(* IEC 61131-3 sources: Std_PalletMover/Class/EncoderpulsesToDegrees, 1 file *)

(* ---- EncoderpulsesToDegrees.st ---- *)
(*!
<Class
	Name               = "EncoderpulsesToDegrees"
	Revision           = "0.0"
	RealtimeTask       = "false"
	CyclicTask         = "true"
	BackgroundTask     = "false"
	Sigmatek           = "false"
	OSInterface        = "false"
	HighPriority       = "false"
	Automatic          = "false"
	UpdateMode         = "Prescan"
	SharedCommandTable = "true"
	Objectsize         = "(512,120)">
	<Channels>
		<Server Name="ClassSvr" Visualized="false" Initialize="false" WriteProtected="true" Retentive="false"/>
		<Server Name="Degrees" Visualized="false" Initialize="false" WriteProtected="true" Retentive="false"/>
		<Server Name="GearRatio" Visualized="false" Initialize="true" WriteProtected="false" Retentive="false"/>
		<Server Name="PulsesPerRound" Visualized="false" Initialize="true" WriteProtected="false" Retentive="false"/>
		<Client Name="EncoderPulses" Required="false" Internal="false"/>
	</Channels>
</Class>
*)
EncoderpulsesToDegrees : CLASS
  //Servers:
	ClassSvr 	: SvrChCmd_DINT;
	PulsesPerRound 	: SvrCh_REAL;
	GearRatio 	: SvrCh_REAL;
	Degrees 	: SvrCh_REAL;
  //Clients:
	EncoderPulses 	: CltCh_DINT;
  //Variables:
  //Functions:

	FUNCTION VIRTUAL GLOBAL CyWork
		VAR_INPUT
			EAX 	: UDINT;
		END_VAR
		VAR_OUTPUT
			state (EAX) 	: UDINT := READY;
		END_VAR;

	FUNCTION VIRTUAL GLOBAL Degrees::Read
		VAR_OUTPUT
			output (EAX) 	: REAL;
		END_VAR;
  //Tables:
	FUNCTION @STD
		VAR_OUTPUT
			ret_code	: CONFSTATES;
		END_VAR;
	FUNCTION GLOBAL TAB @CT_;
END_CLASS;

FUNCTION VIRTUAL GLOBAL EncoderpulsesToDegrees::Degrees::Read
	VAR_OUTPUT
		output (EAX) 	: REAL;
	END_VAR
  VAR
  	realEncoderPulses : REAL;
    tmpDeg            : DINT;
  END_VAR

  EncoderPulses := EncoderPulses.Read();
  realEncoderPulses := to_real(EncoderPulses) - 33236;
  tmpDeg := to_dint(100*realEncoderPulses/GearRatio * (360/PulsesPerRound));
  Degrees := to_real(tmpDeg mod 36000)/100;
	output := Degrees;

END_FUNCTION

FUNCTION VIRTUAL GLOBAL EncoderpulsesToDegrees::CyWork
	VAR_INPUT
		EAX 	: UDINT;
	END_VAR
	VAR_OUTPUT
		state (EAX) 	: UDINT;(* := READY *)
	END_VAR
  VAR
  	realEncoderPulses : REAL;
    tmpDeg            : DINT;
  END_VAR

  EncoderPulses := EncoderPulses.Read();
  realEncoderPulses := to_real(EncoderPulses) - 33236;
  tmpDeg := to_dint(100*realEncoderPulses/GearRatio * (360/PulsesPerRound));
  Degrees := to_real(tmpDeg mod 36000)/100;

END_FUNCTION
